Fanuc KAREL source: kb00034.KL

-- PROVISIONAL review KL for V770-1; original PC SHA256 cd46c539c6a80f24fe9e6addaa31e689b4fb55bd8924c397af1cd3de713c537d
-- Incomplete behavior may be omitted. Consult companion uncertainty JSON. Do not deploy.
PROGRAM KB00034
%NOLOCKGROUP
BEGIN
  -- UNRESOLVED_PC offsets 5-14; opcodes 3F,75
  -- UNRESOLVED_PC offsets 19-37; opcodes 27,22,22,2A,31
  -- UNRESOLVED_PC offsets 42-46; opcodes 7F
END KB00034
